# EPICS IOC start-up script: iocBoot/iocxxx/settings.iocsh
# IOC Title
epicsEnvSet("IOC_NAME", "xxx")

# Logged IOC name for alive and other tools
epicsEnvSet("IOC", "ioc$(IOC_NAME)")

# Shell prompt
epicsEnvSet("IOCSH_PS1", "$(IOC)> ")

# prefix used for all PVs in this IOC
epicsEnvSet("PREFIX", "$(IOC_NAME):")

#For devIocStats
epicsEnvSet("ENGINEER", "engineer")
epicsEnvSet("LOCATION", "$(HOSTNAME=location)")
epicsEnvSet("GROUP", "group")

# search path for database files
epicsEnvSet("EPICS_DB_INCLUDE_PATH", ".:$(TOP)/db")

# search path for streamDevice protocol files
epicsEnvSet("STREAM_PROTOCOL_PATH", ".:$(TOP)/db")

# search path for lua scripts
# epicsEnvSet("LUA_SCRIPT_PATH", "./scripts")

# Specify largest array CA will transport
# Note for N doubles, need N*8 bytes+some overhead
epicsEnvSet("EPICS_CA_MAX_ARRAY_BYTES", 64010)
